// TIA Portal V17 export
// export: Created 2025-03-07T09:19:08.462063Z, ExportSetting WithDefaults, DisplayName Totally Integrated Automation Portal, DisplayVersion V17 Update 8, DisplayName TIA Portal Openness, DisplayVersion V17 Update 8, DisplayName TIA Portal Version Control Interface, DisplayVersion V17, DisplayName SINAMICS Startdrive Advanced, DisplayVersion V17 SP2, DisplayName SINAMICS Startdrive G110M, G120, G120C, G120D, G120P, G115D, DisplayVersion V17 SP2, DisplayName SINAMICS Startdrive G130, G150, S120, S150, SINAMICS MV, S210, DisplayVersion V17 SP2, DisplayName STEP 7 Professional, DisplayVersion V17 Update 8, DisplayName SINUMERIK ONE STEP 7 Toolbox, DisplayVersion V17 Update 12, DisplayName SINUMERIK 840D sl STEP 7 Toolbox, DisplayVersion V17 Update 12, DisplayName STEP 7 Safety, DisplayVersion V17 Update 6, DisplayName WinCC Advanced, DisplayVersion V17 Update 8
DATA_BLOCK "DB10300_PT100_SENSORS_VALUES"   // DB10300
{ S7_Optimized_Access := 'FALSE'; DB_Accessible_From_OPC_UA := 'FALSE' }
VERSION : 0.1
// stored: AutoNumber false, DBAccessibleFromOPCUA false, DBAccessibleFromWebserver true, IsOnlyStoredInLoadMemory false, IsWriteProtectedInAS false
   VAR
      UNIT_01 : Struct
         PT100_SENSOR_1 : Real;   // UNIT 01 PT100 400ºC SENSOR 1
         PT100_SENSOR_2 : Real;   // UNIT 01 PT100 400ºC SENSOR 2
      END_STRUCT;
      UNIT_02 : Struct
         PT100_SENSOR_1 : Real;   // UNIT 02 PT100 400ºC SENSOR 1
         PT100_SENSOR_2 : Real;   // UNIT 02 PT100 400ºC SENSOR 2
      END_STRUCT;
   END_VAR
BEGIN
END_DATA_BLOCK
